// TIA Portal V17 export
// export: Created 2022-01-24T16:28:58.8331874Z, ExportSetting WithDefaults, DisplayName Totally Integrated Automation Portal, DisplayVersion V17, DisplayName TIA Portal Openness, DisplayVersion V17, DisplayName TIA Portal Version Control Interface, DisplayVersion V17, DisplayName SINAMICS Startdrive Advanced, DisplayVersion V17, DisplayName SINAMICS Startdrive G130, G150, S120, S150, SINAMICS MV, S210, DisplayVersion V17, DisplayName SINAMICS Startdrive G110M, G120, G120C, G120D, G120P, G115D, DisplayVersion V17, DisplayName STEP 7 Professional, DisplayVersion V17, DisplayName STEP 7 Safety, DisplayVersion V17, DisplayName WinCC Advanced, DisplayVersion V17
FUNCTION "funkce1" : Void   // FC1, LAD
{ S7_Optimized_Access := 'TRUE' }
AUTHOR : ziz
VERSION : 0.1
// stored: AutoNumber true, IsIECCheckEnabled false, SetENOAutomatically false, UDAEnableTagReadback false
   VAR_INPUT
      cislo1 : Int;
      cislo2 : Int;
   END_VAR
   VAR_OUTPUT
      soucet : Int;
   END_VAR
BEGIN

REGION Network 1
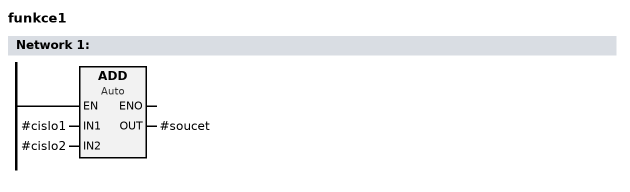
   RUNG wire#powerrail
      Add(in1 := #cislo1, in2 := #cislo2, out => #soucet)
   END_RUNG
   // the same network as SCL:
   #soucet := #cislo1 + #cislo2;
END_REGION
END_FUNCTION
